Universal Robots PolyScope program: calib_poses.urp

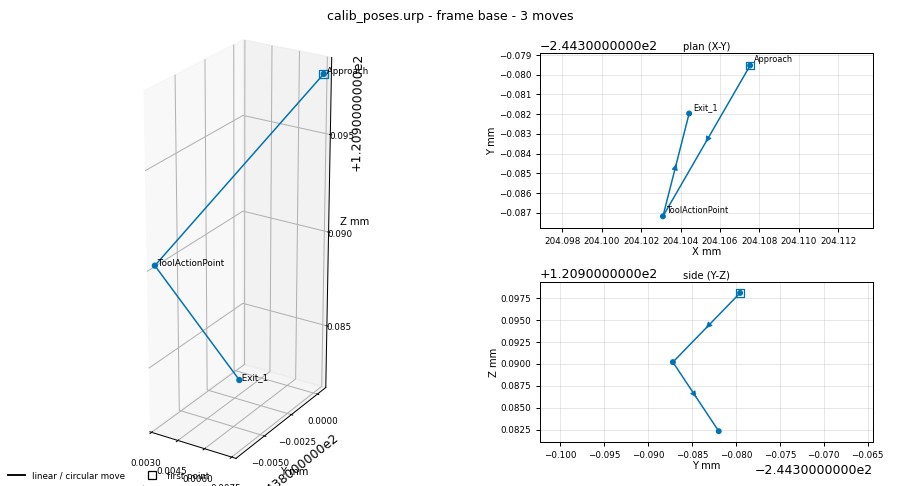
[picture p0: tool path of calib_poses.urp in frame base, 3 of 3 moves have a stored position in this frame; points joined in program order, loops and branches not executed]
Program calib_poses (installation=default directory=/programs/HandEyeCalibration createdIn=3.10.1.76190 lastSavedIn=5.10.0.106288 robotSerialNumber=20185500256)
Calibrated DH parameters: a=[0.000163, -0.146131, -0.38577, 0.000126, -0.000021, 0]; d=[0.161954, 188.306531, -157.478086, -30.695088, 0.099716, 0.099628]; alpha=[1.569701, -0.00212, 0.002263, 1.570438, -1.570123, 0]; deltaTheta=[0, -1.219859, 7.681919, -0.178877, -0.000001, 0]
BeforeStart
  recorder := rpc_factory("xmlrpc", "http://192.168.1.119:10000")
Robot Program (runOnlyOnce=true)
  SuppressedNode
    MoveJ speed 60 deg/s, acceleration 80 deg/s^2 (useActiveTCP=true) feature=Base
      Waypoint Waypoint_2: TCP in base x=367.966 y=-498.532 z=216.454 mm, rx=1.5933 ry=-0.3706 rz=-0.1124 rad; joints [-9.25, -103.416, -103.752, -127.093, 9.101, -16.602] deg; TCP offset x=-0.936 y=-1.83 z=243.679 mm, rx=0 ry=0 rz=0 rad
      Call send_pose
      Waypoint Waypoint_3: TCP in base x=327.963 y=-506.968 z=194.982 mm, rx=1.5932 ry=-0.3708 rz=-0.1124 rad; joints [-11.147, -99.976, -112.479, -115.809, 7.478, -22.644] deg; TCP offset x=-0.936 y=-1.83 z=243.679 mm, rx=0 ry=0 rz=0 rad
      Call send_pose
      Waypoint Waypoint_4: TCP in base x=297.619 y=-506.928 z=194.944 mm, rx=1.5933 ry=-0.3706 rz=-0.1124 rad; joints [-11.949, -96.122, -117.584, -111.122, 6.822, -26.108] deg; TCP offset x=-0.936 y=-1.83 z=243.679 mm, rx=0 ry=0 rz=0 rad
      Call send_pose
      Waypoint Waypoint_5: TCP in base x=228.395 y=-506.957 z=194.993 mm, rx=1.5932 ry=-0.3706 rz=-0.1124 rad; joints [-14.287, -86.954, -130.017, -93.136, 5.131, -40.899] deg; TCP offset x=-0.936 y=-1.83 z=243.679 mm, rx=0 ry=0 rz=0 rad
      Call send_pose
      Waypoint Waypoint_6: TCP in base x=173.626 y=-554.984 z=186.007 mm, rx=1.5835 ry=-0.6041 rz=-0.4205 rad; joints [-25.248, -100.559, -110.469, -120.471, 13.45, -23.039] deg; TCP offset x=-0.936 y=-1.83 z=243.679 mm, rx=0 ry=0 rz=0 rad
      Call send_pose
      Waypoint Waypoint_7: TCP in base x=246.763 y=-390.57 z=166.294 mm, rx=1.8358 ry=0.7613 rz=0.3911 rad; joints [-29.665, -58.875, -131.996, -193.304, -71.061, 3.322] deg; TCP offset x=-0.936 y=-1.83 z=243.679 mm, rx=0 ry=0 rz=0 rad
      Call send_pose
      Waypoint Waypoint_8: TCP in base x=317.855 y=-390.603 z=166.372 mm, rx=1.8358 ry=0.7611 rz=0.3911 rad; joints [-18.47, -66.975, -128.218, -191.178, -60.907, 8.539] deg; TCP offset x=-0.936 y=-1.83 z=243.679 mm, rx=0 ry=0 rz=0 rad
      Call send_pose
      Waypoint Waypoint_9: TCP in base x=407.892 y=-390.567 z=166.317 mm, rx=1.8358 ry=0.7613 rz=0.3911 rad; joints [-11.93, -79.077, -120.342, -188.86, -55.093, 12.052] deg; TCP offset x=-0.936 y=-1.83 z=243.679 mm, rx=0 ry=0 rz=0 rad
      Call send_pose
      Waypoint Waypoint_10: TCP in base x=407.798 y=-483.812 z=189.555 mm, rx=1.598 ry=0.491 rz=0.5731 rad; joints [-27.121, -84.501, -126.95, -153.036, -65.616, 6.599] deg; TCP offset x=-0.936 y=-1.83 z=243.679 mm, rx=0 ry=0 rz=0 rad
      Call send_pose
      Waypoint Waypoint_11: TCP in base x=302.296 y=-483.776 z=189.542 mm, rx=1.598 ry=0.4911 rz=0.5732 rad; joints [-40.29, -74.746, -134.5, -154.86, -78.746, 5.58] deg; TCP offset x=-0.936 y=-1.83 z=243.679 mm, rx=0 ry=0 rz=0 rad
      Call send_pose
      Waypoint Waypoint_12: TCP in base x=302.263 y=-517.38 z=184.021 mm, rx=1.6393 ry=0.1601 rz=0.2686 rad; joints [-21.573, -83.878, -128.517, -154.547, -37.199, 10.201] deg; TCP offset x=-0.936 y=-1.83 z=243.679 mm, rx=0 ry=0 rz=0 rad
      Call send_pose
      Waypoint Waypoint_13: TCP in base x=324.85 y=-440.677 z=177.431 mm, rx=1.6422 ry=0.6272 rz=0.7096 rad; joints [-42.385, -73.276, -134.07, -160.358, -90.617, 6.85] deg; TCP offset x=-0.936 y=-1.83 z=243.679 mm, rx=0 ry=0 rz=0 rad
      Call send_pose
      Waypoint Waypoint_14: TCP in base x=408.664 y=-437.392 z=177.412 mm, rx=1.6422 ry=0.6273 rz=0.7097 rad; joints [-29.678, -79.959, -129.296, -158.689, -78.036, 8.572] deg; TCP offset x=-0.936 y=-1.83 z=243.679 mm, rx=0 ry=0 rz=0 rad
      Call send_pose
      Waypoint Waypoint_15: TCP in base x=408.634 y=-406.103 z=177.456 mm, rx=1.5428 ry=0.9725 rz=0.865 rad; joints [-45.942, -83.113, -124.913, -162.378, -111.937, -1.61] deg; TCP offset x=-0.936 y=-1.83 z=243.679 mm, rx=0 ry=0 rz=0 rad
      Call send_pose
      Waypoint Waypoint_16: TCP in base x=258.316 y=-406.11 z=169.921 mm, rx=1.5101 ry=0.9311 rz=0.9044 rad; joints [-74.693, -81.983, -129.979, -158.37, -140.689, -4.496] deg; TCP offset x=-0.936 y=-1.83 z=243.679 mm, rx=0 ry=0 rz=0 rad
      Call send_pose
      Waypoint Waypoint_17: TCP in base x=258.325 y=-315.913 z=174.16 mm, rx=1.51 ry=0.9312 rz=0.9043 rad; joints [-66.362, -63.996, -140.747, -164.114, -132.486, -2.417] deg; TCP offset x=-0.936 y=-1.83 z=243.679 mm, rx=0 ry=0 rz=0 rad
      Call send_pose
      Waypoint Waypoint_18: TCP in base x=381.314 y=-315.896 z=215.29 mm, rx=1.438 ry=0.9332 rz=0.8818 rad; joints [-32.628, -63.11, -137.141, -163.573, -98.78, 0.148] deg; TCP offset x=-0.936 y=-1.83 z=243.679 mm, rx=0 ry=0 rz=0 rad
      Call send_pose
      Waypoint Waypoint_19: TCP in base x=348.477 y=-484.854 z=193.985 mm, rx=1.7377 ry=0.2177 rz=-0.0301 rad; joints [-9.595, -96.153, -111.343, -187.651, -18.65, 25.465] deg; TCP offset x=-0.936 y=-1.83 z=243.679 mm, rx=0 ry=0 rz=0 rad
      Call send_pose
      Waypoint Waypoint_20: TCP in base x=343.086 y=-510.463 z=285.959 mm, rx=1.5072 ry=-0.3652 rz=0.5041 rad; joints [-12.804, -86.48, -115.361, -151.111, -17.314, 25.154] deg; TCP offset x=-0.936 y=-1.83 z=243.679 mm, rx=0 ry=0 rz=0 rad
      Call send_pose
      Waypoint Waypoint_21: TCP in base x=213.189 y=-570.148 z=273.822 mm, rx=1.6924 ry=-0.7021 rz=-0.4421 rad; joints [-26.201, -99.723, -93.483, -121.533, 19.929, -38.934] deg; TCP offset x=-0.936 y=-1.83 z=243.679 mm, rx=0 ry=0 rz=0 rad
      Call send_pose
      Waypoint Waypoint_22: TCP in base x=213.195 y=-570.121 z=273.84 mm, rx=1.6131 ry=-0.883 rz=-0.5831 rad; joints [-28.293, -110.777, -77.447, -141.342, 27.288, -22.565] deg; TCP offset x=-0.936 y=-1.83 z=243.679 mm, rx=0 ry=0 rz=0 rad
      Call send_pose
      Waypoint Waypoint_23: TCP in base x=170.828 y=-545.037 z=226.414 mm, rx=1.4222 ry=-0.7404 rz=-0.4817 rad; joints [-25.55, -108.999, -95.908, -152.295, 19.783, 7.072] deg; TCP offset x=-0.936 y=-1.83 z=243.679 mm, rx=0 ry=0 rz=0 rad
      Call send_pose
      Waypoint Waypoint_24: TCP in base x=301.867 y=-369.566 z=163.076 mm, rx=1.8743 ry=0.8785 rz=0.395 rad; joints [-21.067, -64.421, -126.968, -198.48, -67.502, 5.881] deg; TCP offset x=-0.936 y=-1.83 z=243.679 mm, rx=0 ry=0 rz=0 rad
      Call send_pose
      Waypoint Waypoint_25: TCP in base x=301.299 y=-522.74 z=264.147 mm, rx=1.3551 ry=-0.2173 rz=0.1611 rad; joints [-15.485, -88.897, -130.052, -96.354, -16.061, -28.882] deg; TCP offset x=-0.936 y=-1.83 z=243.679 mm, rx=0 ry=0 rz=0 rad
      Call send_pose
      Waypoint Waypoint_26: TCP in base x=302.6 y=-435.78 z=239.951 mm, rx=1.8169 ry=-0.102 rz=-0.0971 rad; joints [-2.109, -75.574, -126.691, -87.245, 15.448, -70.568] deg; TCP offset x=-0.936 y=-1.83 z=243.679 mm, rx=0 ry=0 rz=0 rad
      Call send_pose
  Loop Counting (count=24) loopVariable(name=Loop_1)
    URCap Palletizing (polyscope-pallet-impl, Universal Robots) dataModel(palletFeature=Base, isPalletizing=true, Length(key=objectHeight value=0.05 unit=M), Variable(key=name, variable(name=Pallet_1)), Variable(key=globalCountingVariable, variable(name=Pallet_1_cnt, initializeExpression=1)), Variable(key=layerNumberVariable, variable(name=Pallet_1_lno, initializeExpression=1)), Variable(key=layerCountingVariable, variable(name=Pallet_1_lct, initializeExpression=1)), Variable(key=handleSeparatorVariable, variable(name=Pallet_1_sep, initializeExpression=False)), Variable(key=totalCountVariable, variable(name=Pallet_1_tct, initializeExpression=1)), Variable(key=referencePoint, variable(featureName=referencePoint)), Variable(key=separatorPoint, variable(featureName=separatorPoint))); state(isChildrenLocked=true)
      URCap Patterns (polyscope-pallet-impl, Universal Robots) state(isChildrenLocked=true)
        URCap Pattern (polyscope-pallet-impl, Universal Robots) dataModel(UUID=3b75a608-283e-4ba5-887e-097f98334a24, patternType=GRID, rows=6, columns=4, Variable(key=nameVariable, variable(name=Grid_Pattern_1))); state(isChildrenLocked=true)
          URCap Item (polyscope-pallet-impl, Universal Robots) dataModel(UUID=c9c99c67-97d1-430b-a99c-1a147d52fbce, patternType=GRID, index=0, calibrationDeltaTheta=[5.766864417944273E-8, -1.219858784201824, 7.681919015479748, -0.17887715072020058, -5.825955228730417E-7, 1.2463722892999685E-7], calibrationA=[1.6278795868896034E-4, -0.14613148603940784, -0.3857702315473692, 1.264637573695105E-4, -2.1298401427010558E-5, 0.0], calibrationD=[0.16195415116355033, 188.3065313778212, -157.47808565825918, -30.695087710514088, 0.09971634582834017, 0.09962824424434498], calibrationAlpha=[1.5697008015899263, -0.0021197873275575997, 0.0022625217605951827, 1.5704375006736107, -1.570122774022032, 0.0], calibrationJointChecksum=[-1856353559, -1856958578, 625087103, -1528685046, -1528462798, -1527923809], calibrationStatus=2, calibrationValidChecksum=true, baseToFeature=[0.0, 0.0, 0.0, 0.0, 0.0, 0.0], TCPOffset=[-6.811402355588747E-6, -2.240684688920025E-5, 0.25049206407023944, 1.866366297334874E-5, 7.515726035875046E-7, 5.695101542732195E-5], Variable(key=variable, variable(name=CornerItem_1)), JointPositions(key=jointpositions, JointPosition(key=[1], Angle(key=pos value=1.33996 unit=RAD)), JointPosition(key=[2], Angle(key=pos value=-1.250735 unit=RAD)), JointPosition(key=[3], Angle(key=pos value=1.358643 unit=RAD)), JointPosition(key=[4], Angle(key=pos value=-1.180446 unit=RAD)), JointPosition(key=[5], Angle(key=pos value=-1.289172 unit=RAD)), JointPosition(key=[6], Angle(key=pos value=1.586769 unit=RAD))))
          URCap Item (polyscope-pallet-impl, Universal Robots) dataModel(UUID=f56a354f-8c68-413d-8676-7945f6eb2195, patternType=GRID, index=1, calibrationDeltaTheta=[5.766864417944273E-8, -1.219858784201824, 7.681919015479748, -0.17887715072020058, -5.825955228730417E-7, 1.2463722892999685E-7], calibrationA=[1.6278795868896034E-4, -0.14613148603940784, -0.3857702315473692, 1.264637573695105E-4, -2.1298401427010558E-5, 0.0], calibrationD=[0.16195415116355033, 188.3065313778212, -157.47808565825918, -30.695087710514088, 0.09971634582834017, 0.09962824424434498], calibrationAlpha=[1.5697008015899263, -0.0021197873275575997, 0.0022625217605951827, 1.5704375006736107, -1.570122774022032, 0.0], calibrationJointChecksum=[-1856353559, -1856958578, 625087103, -1528685046, -1528462798, -1527923809], calibrationStatus=2, calibrationValidChecksum=true, baseToFeature=[0.0, 0.0, 0.0, 0.0, 0.0, 0.0], TCPOffset=[2.1012148014233623E-5, 5.374124779800038E-6, 0.2504873848051922, -3.637342540473535E-5, -9.132324644629898E-6, -3.138373093022444E-5], Variable(key=variable, variable(name=CornerItem_2)), JointPositions(key=jointpositions, JointPosition(key=[1], Angle(key=pos value=1.836603 unit=RAD)), JointPosition(key=[2], Angle(key=pos value=-0.974145 unit=RAD)), JointPosition(key=[3], Angle(key=pos value=1.103899 unit=RAD)), JointPosition(key=[4], Angle(key=pos value=-1.249341 unit=RAD)), JointPosition(key=[5], Angle(key=pos value=-1.789209 unit=RAD)), JointPosition(key=[6], Angle(key=pos value=3.095536 unit=RAD))))
          URCap Item (polyscope-pallet-impl, Universal Robots) dataModel(UUID=3829da42-c55d-4a5c-b457-f64e555102c7, patternType=GRID, index=2, calibrationDeltaTheta=[5.766864417944273E-8, -1.219858784201824, 7.681919015479748, -0.17887715072020058, -5.825955228730417E-7, 1.2463722892999685E-7], calibrationA=[1.6278795868896034E-4, -0.14613148603940784, -0.3857702315473692, 1.264637573695105E-4, -2.1298401427010558E-5, 0.0], calibrationD=[0.16195415116355033, 188.3065313778212, -157.47808565825918, -30.695087710514088, 0.09971634582834017, 0.09962824424434498], calibrationAlpha=[1.5697008015899263, -0.0021197873275575997, 0.0022625217605951827, 1.5704375006736107, -1.570122774022032, 0.0], calibrationJointChecksum=[-1856353559, -1856958578, 625087103, -1528685046, -1528462798, -1527923809], calibrationStatus=2, calibrationValidChecksum=true, baseToFeature=[0.0, 0.0, 0.0, 0.0, 0.0, 0.0], TCPOffset=[1.176400011337897E-5, -2.5431878820980636E-5, 0.2505117382303935, 6.035514372728441E-5, -1.221505345378224E-7, -7.632465891508638E-6], Variable(key=variable, variable(name=CornerItem_3)), JointPositions(key=jointpositions, JointPosition(key=[1], Angle(key=pos value=2.146494 unit=RAD)), JointPosition(key=[2], Angle(key=pos value=-1.553835 unit=RAD)), JointPosition(key=[3], Angle(key=pos value=1.941673 unit=RAD)), JointPosition(key=[4], Angle(key=pos value=-1.937401 unit=RAD)), JointPosition(key=[5], Angle(key=pos value=-1.951164 unit=RAD)), JointPosition(key=[6], Angle(key=pos value=2.564526 unit=RAD))))
          URCap Item (polyscope-pallet-impl, Universal Robots) dataModel(UUID=a3c91444-18ff-48ff-82e8-cf9579b0eb98, patternType=GRID, index=3, calibrationDeltaTheta=[5.766864417944273E-8, -1.219858784201824, 7.681919015479748, -0.17887715072020058, -5.825955228730417E-7, 1.2463722892999685E-7], calibrationA=[1.6278795868896034E-4, -0.14613148603940784, -0.3857702315473692, 1.264637573695105E-4, -2.1298401427010558E-5, 0.0], calibrationD=[0.16195415116355033, 188.3065313778212, -157.47808565825918, -30.695087710514088, 0.09971634582834017, 0.09962824424434498], calibrationAlpha=[1.5697008015899263, -0.0021197873275575997, 0.0022625217605951827, 1.5704375006736107, -1.570122774022032, 0.0], calibrationJointChecksum=[-1856353559, -1856958578, 625087103, -1528685046, -1528462798, -1527923809], calibrationStatus=2, calibrationValidChecksum=true, baseToFeature=[0.0, 0.0, 0.0, 0.0, 0.0, 0.0], TCPOffset=[-1.5202247894724463E-5, -1.7078883488730323E-5, 0.2504823540438683, 5.8058162637330326E-5, -1.8898539393351993E-5, -4.425319812368838E-5], Variable(key=variable, variable(name=CornerItem_4)), JointPositions(key=jointpositions, JointPosition(key=[1], Angle(key=pos value=0.850612 unit=RAD)), JointPosition(key=[2], Angle(key=pos value=-2.201219 unit=RAD)), JointPosition(key=[3], Angle(key=pos value=2.359599 unit=RAD)), JointPosition(key=[4], Angle(key=pos value=-1.638696 unit=RAD)), JointPosition(key=[5], Angle(key=pos value=-1.177787 unit=RAD)), JointPosition(key=[6], Angle(key=pos value=-0.298551 unit=RAD))))
      URCap Layers (polyscope-pallet-impl, Universal Robots) dataModel(separators=[false], selectedPatterns=[3b75a608-283e-4ba5-887e-097f98334a24])
      URCap At Each Item (polyscope-pallet-impl, Universal Robots) dataModel(selectedPattern=3b75a608-283e-4ba5-887e-097f98334a24, selectedPosition=c9c99c67-97d1-430b-a99c-1a147d52fbce, Approach_calibrationDeltaTheta=[5.766864417944273E-8, -1.219858784201824, 7.681919015479748, -0.17887715072020058, -5.825955228730417E-7, 1.2463722892999685E-7], Approach_calibrationA=[1.6278795868896034E-4, -0.14613148603940784, -0.3857702315473692, 1.264637573695105E-4, -2.1298401427010558E-5, 0.0], Approach_calibrationD=[0.16195415116355033, 188.3065313778212, -157.47808565825918, -30.695087710514088, 0.09971634582834017, 0.09962824424434498], Approach_calibrationAlpha=[1.5697008015899263, -0.0021197873275575997, 0.0022625217605951827, 1.5704375006736107, -1.570122774022032, 0.0], Approach_calibrationJointChecksum=[-1856353559, -1856958578, 625087103, -1528685046, -1528462798, -1527923809], Approach_calibrationStatus=2, Approach_calibrationValidChecksum=true, Approach_baseToFeature=[0.0, 0.0, 0.0, 0.0, 0.0, 0.0], Approach_TCPOffset=[9.452255465045023E-6, -2.9432537538010006E-6, 0.2299935091407426, -7.648093050088842E-6, -1.652261203141786E-5, -3.116940254551279E-5], Exit_calibrationDeltaTheta=[5.766864417944273E-8, -1.219858784201824, 7.681919015479748, -0.17887715072020058, -5.825955228730417E-7, 1.2463722892999685E-7], Exit_calibrationA=[1.6278795868896034E-4, -0.14613148603940784, -0.3857702315473692, 1.264637573695105E-4, -2.1298401427010558E-5, 0.0], Exit_calibrationD=[0.16195415116355033, 188.3065313778212, -157.47808565825918, -30.695087710514088, 0.09971634582834017, 0.09962824424434498], Exit_calibrationAlpha=[1.5697008015899263, -0.0021197873275575997, 0.0022625217605951827, 1.5704375006736107, -1.570122774022032, 0.0], Exit_calibrationJointChecksum=[-1856353559, -1856958578, 625087103, -1528685046, -1528462798, -1527923809], Exit_calibrationStatus=2, Exit_calibrationValidChecksum=true, Exit_baseToFeature=[0.0, 0.0, 0.0, 0.0, 0.0, 0.0], Exit_TCPOffset=[4.545203821995636E-6, 2.318474011053784E-6, 0.2300080487959259, 7.680867283302927E-6, -2.073297310273453E-5, -2.1329974056282276E-5], currentWizardState=LANDING, Pose(key=refBaseToFeature, Position(key=posePosition, Length(key=X value=0 unit=M), Length(key=Y value=0 unit=M), Length(key=Z value=0 unit=M)), Rotation(key=poseRotation, Angle(key=RX value=0 unit=RAD), Angle(key=RY value=0 unit=RAD), Angle(key=RZ value=0 unit=RAD))), Pose(key=refPose, Position(key=posePosition, Length(key=X value=0.204103 unit=M), Length(key=Y value=-0.244387 unit=M), Length(key=Z value=0.12099 unit=M)), Rotation(key=poseRotation, Angle(key=RX value=-2.322256 unit=RAD), Angle(key=RY value=-1.394431 unit=RAD), Angle(key=RZ value=0.21511 unit=RAD))), JointPositions(key=Approach_jointpositions, JointPosition(key=[1], Angle(key=pos value=2.033644 unit=RAD)), JointPosition(key=[2], Angle(key=pos value=-1.618771 unit=RAD)), JointPosition(key=[3], Angle(key=pos value=1.951966 unit=RAD)), JointPosition(key=[4], Angle(key=pos value=-1.487062 unit=RAD)), JointPosition(key=[5], Angle(key=pos value=-1.750784 unit=RAD)), JointPosition(key=[6], Angle(key=pos value=2.562642 unit=RAD))), JointPositions(key=Exit_jointpositions, JointPosition(key=[1], Angle(key=pos value=2.033644 unit=RAD)), JointPosition(key=[2], Angle(key=pos value=-1.618771 unit=RAD)), JointPosition(key=[3], Angle(key=pos value=1.951966 unit=RAD)), JointPosition(key=[4], Angle(key=pos value=-1.487062 unit=RAD)), JointPosition(key=[5], Angle(key=pos value=-1.750784 unit=RAD)), JointPosition(key=[6], Angle(key=pos value=2.562642 unit=RAD))))
        URCap Generated Movements (polyscope-pallet-impl, Universal Robots) state(isChildrenLocked=true)
          MoveJ speed 60 deg/s, acceleration 80 deg/s^2 (useActiveTCP=true) feature=referencePoint
            Waypoint Approach: TCP in base x=204.108 y=-244.38 z=120.998 mm, rx=-2.3222 ry=-1.3945 rz=0.2151 rad; joints [109.519, -84.354, 143.283, -126.372, -103.11, 140.356] deg; TCP offset x=0 y=0 z=0 mm, rx=0 ry=0 rz=0 rad; feature pose in base x=204.103 y=-244.387 z=120.99 mm, rx=-2.3223 ry=-1.3944 rz=0.2151 rad
          MoveL speed 250 mm/s, acceleration 1200 mm/s^2 (useActiveTCP=true) feature(featureName=referencePoint)
            Waypoint ToolActionPoint: TCP in base x=204.103 y=-244.387 z=120.99 mm, rx=-2.3223 ry=-1.3944 rz=0.2151 rad; joints [109.517, -84.352, 143.283, -126.373, -103.11, 140.357] deg; TCP offset x=0 y=0 z=0 mm, rx=0 ry=0 rz=0 rad
          Folder Tool action
            Wait Sleep waitTime=1
            SuppressedNode
              Popup Message (haltProgram=false message=before send inputType=Text)
            Call send_pose
          MoveL speed 250 mm/s, acceleration 1200 mm/s^2 (useActiveTCP=true) feature(featureName=referencePoint)
            Waypoint Exit_1: TCP in base x=204.104 y=-244.382 z=120.982 mm, rx=-2.3222 ry=-1.3945 rz=0.2151 rad; joints [109.518, -84.351, 143.284, -126.375, -103.111, 140.356] deg; TCP offset x=0 y=0 z=0 mm, rx=0 ry=0 rz=0 rad
  SuppressedNode
    Popup Message (haltProgram=false message=before send inputType=Text)
  SuppressedNode
    Call send_pose
SubProgram -> send_pose
SubProgram send_pose (keepSynchronizedWithDisk=false)
  Wait Sleep waitTime=0.5
  Wait Condition expression=is_steady()
  handle := recorder.add_sample(get_actual_tool_flange_pose())
  SuppressedNode
    glob_tcp_pose := get_actual_tcp_pose()
